Fanuc KAREL source: kt00076.KL

-- PROVISIONAL review KL for V1013-1; original PC SHA256 209e3d53934bdb9fa217ad3a24aff4eab6b1b806e10d4652530d247936bc6a36
-- Incomplete behavior may be omitted. Consult companion uncertainty JSON. Do not deploy.
PROGRAM KT00076
%NOLOCKGROUP
VAR
  R1 : REAL
  R2 : REAL
  OUT : REAL
BEGIN
  -- UNRESOLVED_PC offsets 5-16; opcodes 2E,23
  -- UNRESOLVED_PC offsets 21-32; opcodes 2E,23
  -- UNRESOLVED_PC offsets 37-48; opcodes 2E,23
  -- UNRESOLVED_PC offsets 53-64; opcodes 2E,23
  -- UNRESOLVED_PC offsets 69-88; opcodes 21,21,6B,23
  -- UNRESOLVED_PC offsets 93-97; opcodes 7F
END KT00076
